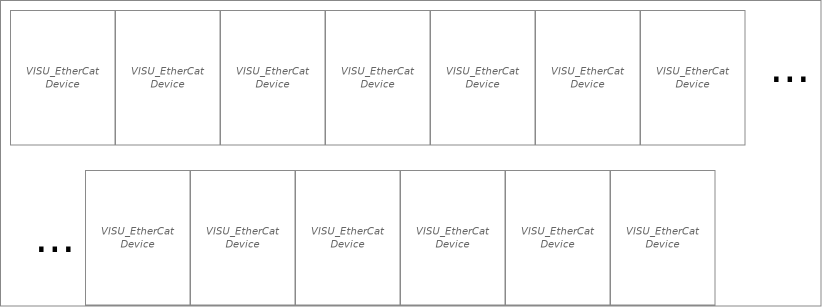
VISUALIZATION VISU_SafetyHydraulicsAndSafetyIO  // 822x307
VAR_IN_OUT
	ref : SafetyHydraulicsAndSafetyIO;
    widget : SafetyHydraulicsAndSafetyIOWidget;
END_VAR
    Frame (10,10 105x135)
        shows VISU_EtherCatDevice(device := ref.parts.COU, widget := widget.COU)
    Frame (115,10 105x135)
        shows VISU_EtherCatDevice(device := ref.parts.DO1, widget := widget.DO1)
    Frame (220,10 105x135)
        shows VISU_EtherCatDevice(device := ref.parts.SI1, widget := widget.SI1)
    Frame (325,10 105x135)
        shows VISU_EtherCatDevice(device := ref.parts.SI2, widget := widget.SI2)
    Frame (535,10 105x135)
        shows VISU_EtherCatDevice(device := ref.parts.SI4, widget := widget.SI4)
    Frame (640,10 105x135)
        shows VISU_EtherCatDevice(device := ref.parts.SL, widget := widget.SL)
    Frame (430,10 105x135)
        shows VISU_EtherCatDevice(device := ref.parts.SI3, widget := widget.SI3)
    Frame (85,170 105x135)
        shows VISU_EtherCatDevice(device := ref.parts.SO1, widget := widget.SO1)
    Label (760,35 60x64), "..."
    Label (25,205 60x64), "..."
    Frame (190,170 105x135)
        shows VISU_EtherCatDevice(device := ref.parts.AI1, widget := widget.AI1)
    Frame (295,170 105x135)
        shows VISU_EtherCatDevice(device := ref.parts.AI2, widget := widget.AI2)
    Frame (400,170 105x135)
        shows VISU_EtherCatDevice(device := ref.parts.RTD1, widget := widget.RTD1)
    Frame (505,170 105x135)
        shows VISU_EtherCatDevice(device := ref.parts.PWR1, widget := widget.PWR1)
    Frame (610,170 105x135)
        shows VISU_EtherCatDevice(device := ref.parts.AO1, widget := widget.AO1)
END_VISUALIZATION

(* stored: Version 1.1.0.1, ProductVersion 3.1.4019.2
   Visu VISU_SafetyHydraulicsAndSafetyIO: Id {e22a28c2-0238-4515-9240-b8ab476c5d4c} *)
